TYPE ST_Outputs :
STRUCT
	// To controller
	fWref 					AT %Q*				: LREAL;
	fWactual 				AT %Q*				: LREAL;
	fWmech					AT %Q* 				: LREAL;
	fIa, fIb, fIc 			AT %Q*				: LREAL;
	fTcTheta				AT %Q*				: LREAL;
	fThetaMech 				AT %Q* 				: LREAL;
	fControlEnable 			AT %Q*				: LREAL := 0;
	// CAN
	Outputs					AT %Q*				: CANTXQUEUESTRUCT_N_1;
	// Encoder
	uEL5101_CounterSet 		AT %Q*				: UINT;
	uEL5101_CounterSetWORD 	AT %Q* 				: WORD;
END_STRUCT
END_TYPE

(* stored: Version 1.1.0.1, ProductVersion 3.1.4024.11
   DUT ST_Outputs: Id {d85eb51e-193b-4311-b97f-7f95096a0309} *)
